// TIA Portal project "factory_io_from_a2b_set_and_reset" (V19)

(* hardware
DEVICE "S7-1200 station_1"  S7-1200 Station
   slot 0: "Rack_0"  S7-1200 Rack  Rack  V1.0
   slot 1: "PLC_1"  CPU 1212C DC/DC/Rly  6ES7 212-1HE40-0XB0  V4.5
*)

// ===== PLC "PLC_1"  CPU 1212C DC/DC/Rly =====

VAR_GLOBAL   // PLC tag table "Default tag table"
   "Start" AT %I0.2 : Bool;
   "Sensor1" AT %I0.0 : Bool;
   "Sensor2" AT %I0.1 : Bool;
   "Conveyor" AT %Q0.0 : Bool;
   "Entry Conveyor" AT %Q0.1 : Bool;
   "Conveyor Reset" AT %M0.1 : Bool;
   "Conveyor Set" AT %M0.0 : Bool;
   "Reset" AT %I0.3 : Bool;
END_VAR

ORGANIZATION_BLOCK "Main"   // OB1, LAD, ProgramCycle
TITLE = "Main Program Sweep (Cycle)"
{ S7_Optimized_Access := 'TRUE' }
VERSION : 0.1
   VAR_INPUT
      Initial_Call : Bool;   // Initial call of this OB
      Remanence : Bool;   // =True, if remanent data are available
   END_VAR
BEGIN

REGION Network 1
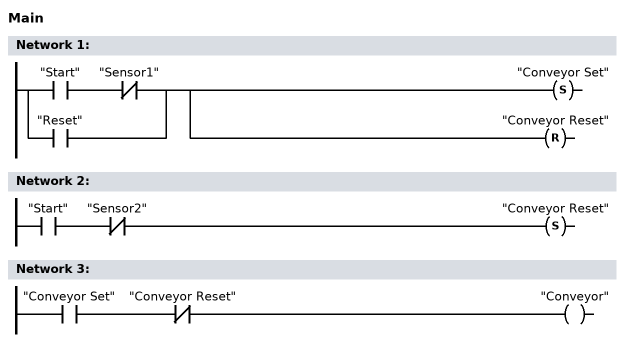
   RUNG wire#powerrail
      Contact( "Start" )
      I_Contact( "Sensor1" )
      wire#w1
      S_Coil( "Conveyor Set" )
   END_RUNG
   RUNG wire#powerrail
      Contact( "Reset" )
   END_RUNG wire#w1
   RUNG wire#w1
      R_Coil( "Conveyor Reset" )
   END_RUNG
   // the same network as SCL:
   IF ("Start" AND NOT "Sensor1") OR "Reset" THEN
       "Conveyor Set" := TRUE;
       "Conveyor Reset" := FALSE;
   END_IF;
END_REGION

REGION Network 2
   RUNG wire#powerrail
      Contact( "Start" )
      I_Contact( "Sensor2" )
      S_Coil( "Conveyor Reset" )
   END_RUNG
   // the same network as SCL:
   IF "Start" AND NOT "Sensor2" THEN "Conveyor Reset" := TRUE; END_IF;
END_REGION

REGION Network 3
   RUNG wire#powerrail
      Contact( "Conveyor Set" )
      I_Contact( "Conveyor Reset" )
      Coil( "Conveyor" )
   END_RUNG
   // the same network as SCL:
   "Conveyor" := "Conveyor Set" AND NOT "Conveyor Reset";
END_REGION
END_ORGANIZATION_BLOCK